(* IEC 61131-3 sources: plc-agent/tests/fixtures/p3_small, 1 file *)

(* ---- Main.st ---- *)
PROGRAM MAIN
VAR
    StartPB AT %IX0.0 : BOOL;
    Motor AT %QX0.0 : BOOL;
END_VAR
Motor := StartPB;
END_PROGRAM
